FUNCTION FUN_RangeOutside : BOOL
VAR_INPUT
	fValue		:REAL;			// Actual value
	fLimitHigh	:REAL;			// High limit for range
	fLimitLow	:REAL;			// Low limit for range
END_VAR
VAR_OUTPUT
	bHigh		:BOOL;			// True if value is greater than rLimitHigh
	bLow		:BOOL;			// True if value is lower than rLimitLow	
END_VAR
VAR
	bOutside	:BOOL;			// True if value is outside of range
END_VAR


// Compare actual value with range
IF fValue < fLimitLow OR fValue > fLimitHigh THEN
	// Outside range
	bOutside := TRUE;
	IF fValue > fLimitHigh THEN
		bHigh := TRUE;
		bLow := FALSE;
	ELSE
		bHigh := FALSE;
		bLow := TRUE;
	END_IF
ELSE
	// Inside of range
	bOutside := FALSE;
END_IF

// Set return value
FUN_RangeOutside := bOutside;

END_FUNCTION

(* stored: Version 1.1.0.1, ProductVersion 3.1.4024.12
   POU FUN_RangeOutside: Id {9517141a-21c8-4fa0-943b-f38964dbf8f3}, SpecialFunc None *)
